Staubli VAL3: speedCase0_15.pgx

program speedCase0_15(num x_nNum (dimensions=1))
begin
  switch x_nNum
    case 0
      dioSet(doB_0_speed,0)
      dioSet(doB_1_speed,0)
      dioSet(doB_2_speed,0)
      dioSet(doB_3_speed,0)
      dioSet(doB_4_speed,0)
      dioSet(doB_5_speed,0)
    break
    case 1
      dioSet(doB_0_speed,1)
      dioSet(doB_1_speed,0)
      dioSet(doB_2_speed,0)
      dioSet(doB_3_speed,0)
      dioSet(doB_4_speed,0)
      dioSet(doB_5_speed,0)
    break
    case 2
      dioSet(doB_1_speed,1)
      dioSet(doB_0_speed,0)
      dioSet(doB_2_speed,0)
      dioSet(doB_3_speed,0)
      dioSet(doB_4_speed,0)
      dioSet(doB_5_speed,0)
    break
    case 3
      dioSet(doB_0_speed,1)
      dioSet(doB_1_speed,1)
      dioSet(doB_2_speed,0)
      dioSet(doB_3_speed,0)
      dioSet(doB_4_speed,0)
      dioSet(doB_5_speed,0)
    break
    case 4
      dioSet(doB_2_speed,1)
      dioSet(doB_0_speed,0)
      dioSet(doB_1_speed,0)
      dioSet(doB_3_speed,0)
      dioSet(doB_4_speed,0)
      dioSet(doB_5_speed,0)
    break
    case 5
      dioSet(doB_0_speed,1)
      dioSet(doB_2_speed,1)
      dioSet(doB_1_speed,0)
      dioSet(doB_3_speed,0)
      dioSet(doB_4_speed,0)
      dioSet(doB_5_speed,0)
    break
    case 6
      dioSet(doB_1_speed,1)
      dioSet(doB_2_speed,1)
      dioSet(doB_0_speed,0)
      dioSet(doB_3_speed,0)
      dioSet(doB_4_speed,0)
      dioSet(doB_5_speed,0)
    break
    case 7
      dioSet(doB_0_speed,1)
      dioSet(doB_1_speed,1)
      dioSet(doB_2_speed,1)
      dioSet(doB_3_speed,0)
      dioSet(doB_4_speed,0)
      dioSet(doB_5_speed,0)
    break

    case 8
      dioSet(doB_3_speed,1)
      dioSet(doB_0_speed,0)
      dioSet(doB_1_speed,0)
      dioSet(doB_2_speed,0)
      dioSet(doB_4_speed,0)
      dioSet(doB_5_speed,0)
    break
    case 9
      dioSet(doB_0_speed,1)
      dioSet(doB_1_speed,0)
      dioSet(doB_2_speed,0)
      dioSet(doB_3_speed,1)
      dioSet(doB_4_speed,0)
      dioSet(doB_5_speed,0)
    break
    case 10
      dioSet(doB_1_speed,1)
      dioSet(doB_0_speed,0)
      dioSet(doB_3_speed,1)
      dioSet(doB_2_speed,0)
      dioSet(doB_4_speed,0)
      dioSet(doB_5_speed,0)
    break
    case 11
      dioSet(doB_0_speed,1)
      dioSet(doB_1_speed,1)
      dioSet(doB_3_speed,1)
      dioSet(doB_2_speed,0)
      dioSet(doB_4_speed,0)
      dioSet(doB_5_speed,0)
    break
    case 12
      dioSet(doB_2_speed,1)
      dioSet(doB_3_speed,1)
      dioSet(doB_0_speed,0)
      dioSet(doB_1_speed,0)
      dioSet(doB_4_speed,0)
      dioSet(doB_5_speed,0)
    break
    case 13
      dioSet(doB_0_speed,1)
      dioSet(doB_2_speed,1)
      dioSet(doB_3_speed,1)
      dioSet(doB_1_speed,0)
      dioSet(doB_4_speed,0)
      dioSet(doB_5_speed,0)
    break
    case 14
      dioSet(doB_1_speed,1)
      dioSet(doB_2_speed,1)
      dioSet(doB_3_speed,1)
      dioSet(doB_0_speed,0)
      dioSet(doB_4_speed,0)
      dioSet(doB_5_speed,0)
    break
    case 15
      dioSet(doB_0_speed,1)
      dioSet(doB_1_speed,1)
      dioSet(doB_2_speed,1)
      dioSet(doB_3_speed,1)
      dioSet(doB_4_speed,0)
      dioSet(doB_5_speed,0)
    break
  endSwitch
end
